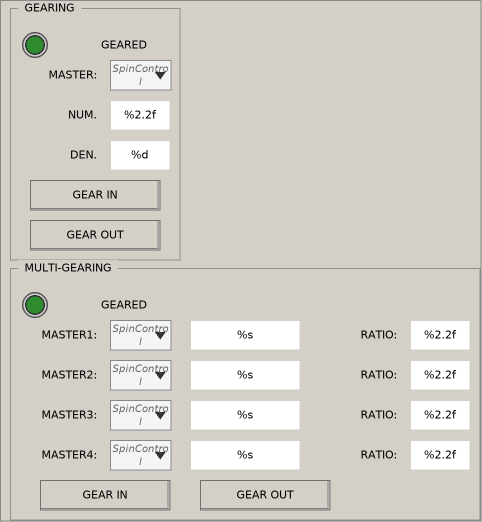
VISUALIZATION Gearing  // 482x522
    GroupBox (10,0 170x260), "GEARING"
        Textfield (40,30 100x30), "GEARED", text variable: MAIN.hmiAxisSelect
        SpinControl (100,60 61x30), variable: GVL.axes[MAIN.hmiAxisSelect].masterAxis
            p651134158: GVL.axisNumMax
            OnMouseClick: write GVL.axes[MAIN.hmiAxisSelect].masterAxis via Default
        Textfield (10,60 80x30), "MASTER:", text variable: MAIN.hmiAxisSelect
        Textfield (100,100 60x30), "%2.2f", text variable: GVL.axes[MAIN.hmiAxisSelect].fGearRatioNum
            OnMouseClick: write GVL.axes[MAIN.hmiAxisSelect].fGearRatioNum via Default
        Textfield (10,100 80x30), "NUM.", text variable: MAIN.hmiAxisSelect
        Textfield (100,140 60x30), "%d", text variable: GVL.axes[MAIN.hmiAxisSelect].iGearRatioDen
            OnMouseClick: write GVL.axes[MAIN.hmiAxisSelect].iGearRatioDen via Default
        Textfield (10,140 80x30), "DEN.", text variable: MAIN.hmiAxisSelect
        Button (20,180 130x30), "GEAR IN"
            OnMouseClick: execute { GVL.axes[MAIN.hmiAxisSelect].eCommand:=eMcCommand.GearIn; GVL.axes[MAIN.hmiAxisSelect].bExecute:= TRUE; }
        Button (20,220 130x30), "GEAR OUT"
            OnMouseClick: execute { GVL.axes[MAIN.hmiAxisSelect].eCommand:=eMcCommand.GearOut; GVL.axes[MAIN.hmiAxisSelect].bExecute:= TRUE; }
        Lamp1 (10,30 30x30), variable: GVL.axes[MAIN.hmiAxisSelect].iAxisState=500, style: Lamp-Lamp1-Green
    GroupBox (10,260 470x260), "MULTI-GEARING"
        Lamp1 (10,30 30x30), variable: GVL.axes[MAIN.hmiAxisSelect].iAxisState=500, style: Lamp-Lamp1-Green
        Textfield (40,30 100x30), "GEARED", text variable: MAIN.hmiAxisSelect
        SpinControl (100,60 61x30), variable: GVL.axes[MAIN.hmiAxisSelect].masterAxes[1].i
            p651134158: GVL.axisNumMax
            OnMouseClick: write GVL.axes[MAIN.hmiAxisSelect].masterAxes[1].i via Default
        Textfield (10,60 80x30), "MASTER1:", text variable: MAIN.hmiAxisSelect
        Textfield (400,60 60x30), "%2.2f", text variable: GVL.axes[MAIN.hmiAxisSelect].masterAxes[1].ratio
            OnMouseClick: write GVL.axes[MAIN.hmiAxisSelect].masterAxes[1].ratio via Default
        Textfield (310,60 80x30), "RATIO:", text variable: MAIN.hmiAxisSelect
        Button (30,220 130x30), "GEAR IN"
            OnMouseClick: execute { GVL.axes[MAIN.hmiAxisSelect].eCommand:=eMcCommand.GearInMultiMaster; GVL.axes[MAIN.hmiAxisSelect].bExecute:= TRUE; }
        Button (190,220 130x30), "GEAR OUT"
            OnMouseClick: execute { GVL.axes[MAIN.hmiAxisSelect].eCommand:=eMcCommand.GearOut; GVL.axes[MAIN.hmiAxisSelect].bExecute:= TRUE; }
        SpinControl (100,100 61x30), variable: GVL.axes[MAIN.hmiAxisSelect].masterAxes[2].i
            p651134158: GVL.axisNumMax
            OnMouseClick: write GVL.axes[MAIN.hmiAxisSelect].masterAxes[2].i via Default
        SpinControl (100,140 61x30), variable: GVL.axes[MAIN.hmiAxisSelect].masterAxes[3].i
            p651134158: GVL.axisNumMax
            OnMouseClick: write GVL.axes[MAIN.hmiAxisSelect].masterAxes[3].i via Default
        SpinControl (100,180 61x30), variable: GVL.axes[MAIN.hmiAxisSelect].masterAxes[4].i
            p651134158: GVL.axisNumMax
            OnMouseClick: write GVL.axes[MAIN.hmiAxisSelect].masterAxes[4].i via Default
        Textfield (310,100 80x30), "RATIO:", text variable: MAIN.hmiAxisSelect
        Textfield (310,140 80x30), "RATIO:", text variable: MAIN.hmiAxisSelect
        Textfield (310,180 80x30), "RATIO:", text variable: MAIN.hmiAxisSelect
        Textfield (10,100 80x30), "MASTER2:", text variable: MAIN.hmiAxisSelect
        Textfield (10,140 80x30), "MASTER3:", text variable: MAIN.hmiAxisSelect
        Textfield (10,180 80x30), "MASTER4:", text variable: MAIN.hmiAxisSelect
        Textfield (400,100 60x30), "%2.2f", text variable: GVL.axes[MAIN.hmiAxisSelect].masterAxes[2].ratio
            OnMouseClick: write GVL.axes[MAIN.hmiAxisSelect].masterAxes[2].ratio via Default
        Textfield (400,140 60x30), "%2.2f", text variable: GVL.axes[MAIN.hmiAxisSelect].masterAxes[3].ratio
            OnMouseClick: write GVL.axes[MAIN.hmiAxisSelect].masterAxes[3].ratio via Default
        Textfield (400,180 60x30), "%2.2f", text variable: GVL.axes[MAIN.hmiAxisSelect].masterAxes[4].ratio
            OnMouseClick: write GVL.axes[MAIN.hmiAxisSelect].masterAxes[4].ratio via Default
        Textfield (180,60 110x30), "%s", text variable: GVL.axes[GVL.axes[MAIN.hmiAxisSelect].masterAxes[1].i].sAxisName
        Textfield (180,100 110x30), "%s", text variable: GVL.axes[GVL.axes[MAIN.hmiAxisSelect].masterAxes[2].i].sAxisName
        Textfield (180,140 110x30), "%s", text variable: GVL.axes[GVL.axes[MAIN.hmiAxisSelect].masterAxes[3].i].sAxisName
        Textfield (180,180 110x30), "%s", text variable: GVL.axes[GVL.axes[MAIN.hmiAxisSelect].masterAxes[4].i].sAxisName
END_VISUALIZATION

(* stored: Version 1.1.0.1, ProductVersion 3.1.4022.12
   Visu Gearing: Id {2b912947-8f75-4479-907b-17dd521d3090} *)
